FUNCTION_BLOCK EL3612
VAR
	_io : EL36x2_Data;
	{attribute addProperty Name "WcState"}
	_wcState : WcStateInputToggle;
	{attribute addProperty Name "Info data"}
	_infoData : InfoDataAds;
END_VAR

PROPERTY IO : REFERENCE TO EL36x2_Data
GET
IO REF= _io;
END_GET
END_PROPERTY

PROPERTY WcState : REFERENCE TO WcStateInputToggle
GET
WcState REF= _wcState;
END_GET
END_PROPERTY

END_FUNCTION_BLOCK

(* stored: Version 1.1.0.1, ProductVersion 3.1.4024.9
   POU EL3612: Id {02eb6413-1036-004a-29b4-ab09b84d237b}, SpecialFunc None
   Property IO: Id {4793406c-040e-0533-345e-434e433fa568}
   Get Get: Id {c5af9bcc-9972-07b2-2be6-17b488a3c550}
   Property WcState: Id {819d421f-94e7-002d-3b2d-e63eec09bdd2}
   Get Get: Id {9f26aaba-9446-03ff-3a9d-a2be2520cf67} *)
